(* IEC 61131-3 sources: Summary-ETFA22/ahorn/benchmark/PPU/Scenario3v1_Final, 6 files *)

(* ---- Scenario3v1_Final_Type.st ---- *)
TYPE
    Stamp_states_t : (Green_Lamp , Init , Interstep , Interstep_2 , StampProcess , StampSliderBack , StampSliderForward , Stamp_Init_1 , Stamp_Init_2 , Stamp_Init_3 , Stamp_Init_4 , Start_Stamp , Step0 , Step1 , Step2);
    Magazin_states_t : (Green_Lamp , Init , Interstep , Magazin_Init , Magazin_Init_2 , Slider_Move_Back , Start_Magazin , Step0 , Step1 , convey);
    Crane_states_t : (Crane_Go_Up , Crane_Init , Crane_Init_2 , Crane_Lift_At_Stamp , Crane_Lift_Conveyor , Crane_Lift_Magazin , Crane_Lift_Magazin_Metallic , Crane_Lower , Crane_On_Conveyor , Crane_On_Conveyor_Metallic , Crane_On_Stamp_Metallic , Crane_Turn_Left_From_Stamp , Crane_Turn_Left_Metallic , Crane_Turn_Left_NOT_Metallic , Init , Interstep , Interstep_2 , Interstep_Check_Workpiece , Lower_Crane , Reset_interconnect , Start_Crane , Step0 , Step2 , Suck_At_Stamp , TimeDelay , Turn_Right , Wait_At_Stamp , pause , release , release_Workpiece);
END_TYPE

(* ---- Scenario3v1_Final_Crane.st ---- *)
FUNCTION_BLOCK Crane
    VAR_INPUT  CraneDown : BOOL; END_VAR
    VAR_OUTPUT  CraneLower : BOOL; END_VAR
    VAR_INPUT  CraneOnConveyor : BOOL; END_VAR
    VAR_INPUT  CraneOnMagazin : BOOL; END_VAR
    VAR_INPUT  CranePositionStamp : BOOL; END_VAR
    VAR_INPUT  CraneSucked : BOOL; END_VAR
    VAR_OUTPUT  CraneTurnClockwise : BOOL; END_VAR
    VAR_OUTPUT  CraneTurnCounterclockwise : BOOL; END_VAR
    VAR_INPUT  CraneUp : BOOL; END_VAR
    VAR  Duration1 : TIME := TIME#1s500.0ms; END_VAR
    VAR_INPUT  MagazinCapacitiveSensor : BOOL; END_VAR
    VAR_OUTPUT  MagazinVacuumOff : BOOL; END_VAR
    VAR_OUTPUT  MagazinVacuumOn : BOOL; END_VAR
    VAR  SFCInit : BOOL; END_VAR
    VAR_INPUT  SFCReset : BOOL; END_VAR
    VAR_INPUT  SliderMovedOut : BOOL; END_VAR
    VAR_INPUT  SliderNotMovedOut : BOOL; END_VAR
    VAR_INPUT  StampLowered : BOOL; END_VAR
    VAR_INPUT  StampSliderFilled : BOOL; END_VAR
    VAR_INPUT  StartButtonMagazin : BOOL; END_VAR
    VAR_OUTPUT  StartCommandCrane : BOOL; END_VAR
    VAR_INPUT  StartVar : BOOL; END_VAR
    VAR  TimeDelay_Timer : TON; END_VAR
    VAR  TimeDelay_Timer_Duration : TIME := TIME#50.0ms; END_VAR
    VAR  TimeDelay_Timer_interconnect : BOOL; END_VAR
    VAR  Timer1 : TON; END_VAR
    VAR_INPUT  WorkpieceReady : BOOL; END_VAR
    VAR  State : Crane_states_t; END_VAR
    VAR  Transit : BOOL; END_VAR
    VAR  actualtime1 : TIME; END_VAR
    VAR  interconnect : BOOL; END_VAR
    VAR  interconnectCraneStartCommand : BOOL; END_VAR

    CASE State OF
        Crane_states_t#Crane_Go_Up:
            Transit := FALSE;
            CraneLower := FALSE;
            IF CraneUp THEN
                Transit := TRUE;
                State := Crane_states_t#pause;
            END_IF;

        Crane_states_t#Crane_Init:
            Transit := FALSE;
            CraneLower := TRUE;
            interconnectCraneStartCommand := FALSE;
            IF CraneDown THEN
                Transit := TRUE;
                State := Crane_states_t#Crane_Init_2;
            END_IF;

        Crane_states_t#Crane_Init_2:
            Transit := FALSE;
            CraneLower := FALSE;
            IF CraneUp THEN
                Transit := TRUE;
                State := Crane_states_t#Interstep;
            END_IF;

        Crane_states_t#Crane_Lift_At_Stamp:
            Transit := FALSE;
            CraneLower := FALSE;
            IF CraneUp THEN
                Transit := TRUE;
                State := Crane_states_t#Crane_Turn_Left_From_Stamp;
            END_IF;

        Crane_states_t#Crane_Lift_Conveyor:
            Transit := FALSE;
            CraneLower := FALSE;
            IF TRUE THEN
                Transit := TRUE;
                State := Crane_states_t#Interstep;
            END_IF;

        Crane_states_t#Crane_Lift_Magazin:
            Transit := FALSE;
            CraneLower := FALSE;
            IF CraneUp THEN
                Transit := TRUE;
                State := Crane_states_t#Crane_Turn_Left_NOT_Metallic;
            END_IF;

        Crane_states_t#Crane_Lift_Magazin_Metallic:
            Transit := FALSE;
            CraneLower := FALSE;
            IF CraneUp THEN
                Transit := TRUE;
                State := Crane_states_t#Crane_Turn_Left_Metallic;
            END_IF;

        Crane_states_t#Crane_Lower:
            Transit := FALSE;
            MagazinVacuumOn := TRUE;
            MagazinVacuumOff := FALSE;
            CraneLower := TRUE;
            IF CraneSucked THEN
                Transit := TRUE;
                State := Crane_states_t#Step0;
            END_IF;

        Crane_states_t#Crane_On_Conveyor:
            Transit := FALSE;
            CraneTurnCounterclockwise := FALSE;
            CraneTurnClockwise := FALSE;
            CraneLower := TRUE;
            IF CraneDown THEN
                Transit := TRUE;
                State := Crane_states_t#release;
            END_IF;

        Crane_states_t#Crane_On_Conveyor_Metallic:
            Transit := FALSE;
            CraneTurnCounterclockwise := FALSE;
            CraneTurnClockwise := FALSE;
            CraneLower := TRUE;
            IF CraneDown THEN
                Transit := TRUE;
                State := Crane_states_t#release;
            END_IF;

        Crane_states_t#Crane_On_Stamp_Metallic:
            Transit := FALSE;
            CraneTurnCounterclockwise := FALSE;
            CraneTurnClockwise := FALSE;
            CraneLower := TRUE;
            IF CraneDown THEN
                Transit := TRUE;
                State := Crane_states_t#release_Workpiece;
            END_IF;

        Crane_states_t#Crane_Turn_Left_From_Stamp:
            Transit := FALSE;
            CraneTurnClockwise := TRUE;
            CraneTurnCounterclockwise := FALSE;
            IF CraneOnConveyor THEN
                Transit := TRUE;
                State := Crane_states_t#Crane_On_Conveyor_Metallic;
            END_IF;

        Crane_states_t#Crane_Turn_Left_Metallic:
            Transit := FALSE;
            CraneTurnCounterclockwise := TRUE;
            CraneTurnClockwise := FALSE;
            IF CranePositionStamp THEN
                Transit := TRUE;
                State := Crane_states_t#Crane_On_Stamp_Metallic;
            END_IF;

        Crane_states_t#Crane_Turn_Left_NOT_Metallic:
            Transit := FALSE;
            CraneTurnCounterclockwise := TRUE;
            CraneTurnClockwise := FALSE;
            IF CraneOnConveyor THEN
                Transit := TRUE;
                State := Crane_states_t#Crane_On_Conveyor;
            END_IF;

        Crane_states_t#Init:
            Transit := FALSE;
            IF TRUE THEN
                Transit := TRUE;
                State := Crane_states_t#Start_Crane;
            END_IF;

        Crane_states_t#Interstep:
            Transit := FALSE;
            StartCommandCrane := TRUE;
            IF StartVar THEN
                Transit := TRUE;
                State := Crane_states_t#Interstep_2;
            END_IF;

        Crane_states_t#Interstep_2:
            Transit := FALSE;
            IF SliderMovedOut THEN
                Transit := TRUE;
                State := Crane_states_t#TimeDelay;
            END_IF;

        Crane_states_t#Interstep_Check_Workpiece:
            Transit := FALSE;
            CraneTurnClockwise := FALSE;
            CraneTurnCounterClockwise := FALSE;
            IF WorkpieceReady THEN
                Transit := TRUE;
                State := Crane_states_t#Crane_Lower;
            ELSIF (NOT WorkpieceReady AND NOT StampSliderFilled) THEN
                Transit := TRUE;
                State := Crane_states_t#Step2;
            ELSIF (NOT WorkpieceReady AND StampSliderFilled) THEN
                Transit := TRUE;
                State := Crane_states_t#Wait_At_Stamp;
            END_IF;

        Crane_states_t#Lower_Crane:
            Transit := FALSE;
            CraneLower := TRUE;
            IF CraneDown THEN
                Transit := TRUE;
                State := Crane_states_t#Suck_At_Stamp;
            END_IF;

        Crane_states_t#Reset_interconnect:
            Transit := FALSE;
            interconnect := FALSE;
            Timer1(IN := FALSE, PT := TIME#1.0ms);
            IF SliderMovedOut THEN
                Transit := TRUE;
                State := Crane_states_t#Lower_Crane;
            END_IF;

        Crane_states_t#Start_Crane:
            Transit := FALSE;
            CraneLower := FALSE;
            MagazinVacuumOff := TRUE;
            MagazinVacuumOn := FALSE;
            CraneTurnCounterclockwise := FALSE;
            CraneTurnClockwise := FALSE;
            StartVar := FALSE;
            StartCommandCrane := FALSE;
            IF (StartButtonMagazin = TRUE) THEN
                interconnectCraneStartCommand := TRUE;
            END_IF;
            IF interconnectCraneStartCommand THEN
                Transit := TRUE;
                State := Crane_states_t#Crane_Init;
            END_IF;

        Crane_states_t#Step0:
            Transit := FALSE;
            IF NOT MagazinCapacitiveSensor THEN
                Transit := TRUE;
                State := Crane_states_t#Crane_Lift_Magazin;
            ELSIF MagazinCapacitiveSensor THEN
                Transit := TRUE;
                State := Crane_states_t#Crane_Lift_Magazin_Metallic;
            END_IF;

        Crane_states_t#Step2:
            Transit := FALSE;
            IF TRUE THEN
                Transit := TRUE;
                State := Crane_states_t#Start_Crane;
            END_IF;

        Crane_states_t#Suck_At_Stamp:
            Transit := FALSE;
            MagazinVacuumOn := TRUE;
            MagazinVacuumOff := FALSE;
            IF CraneSucked THEN
                Transit := TRUE;
                State := Crane_states_t#Crane_Lift_At_Stamp;
            END_IF;

        Crane_states_t#TimeDelay:
            Transit := FALSE;
            TimeDelay_Timer(IN := TRUE, PT := TimeDelay_Timer_Duration);
            TimeDelay_Timer_interconnect := TimeDelay_Timer.Q;
            IF TimeDelay_Timer_interconnect THEN
                Transit := TRUE;
                State := Crane_states_t#Turn_Right;
            END_IF;

        Crane_states_t#Turn_Right:
            Transit := FALSE;
            CraneTurnClockwise := TRUE;
            CraneTurnCounterclockwise := FALSE;
            IF CraneOnMagazin THEN
                Transit := TRUE;
                State := Crane_states_t#Interstep_Check_Workpiece;
            END_IF;

        Crane_states_t#Wait_At_Stamp:
            Transit := FALSE;
            IF TRUE THEN
                Transit := TRUE;
                State := Crane_states_t#pause;
            END_IF;

        Crane_states_t#pause:
            Transit := FALSE;
            Timer1(IN := CraneUp, PT := Duration1);
            interconnect := Timer1.Q;
            IF interconnect THEN
                Transit := TRUE;
                State := Crane_states_t#Reset_interconnect;
            END_IF;

        Crane_states_t#release:
            Transit := FALSE;
            MagazinVacuumOff := TRUE;
            MagazinVacuumOn := FALSE;
            IF TRUE THEN
                Transit := TRUE;
                State := Crane_states_t#Crane_Lift_Conveyor;
            END_IF;

        Crane_states_t#release_Workpiece:
            Transit := FALSE;
            MagazinVacuumOff := TRUE;
            MagazinVacuumOn := FALSE;
            IF TRUE THEN
                Transit := TRUE;
                State := Crane_states_t#Crane_Go_Up;
            END_IF;
    END_CASE;
END_FUNCTION_BLOCK

(* ---- Scenario3v1_Final_Magazin.st ---- *)
FUNCTION_BLOCK Magazin
    VAR_INPUT  CraneDown : BOOL; END_VAR
    VAR_OUTPUT  CraneLower : BOOL; END_VAR
    VAR_INPUT  CraneOnConveyor : BOOL; END_VAR
    VAR_INPUT  CraneOnMagazin : BOOL; END_VAR
    VAR_INPUT  CraneSucked : BOOL; END_VAR
    VAR_OUTPUT  CraneTurnClockwise : BOOL; END_VAR
    VAR_OUTPUT  CraneTurnCounterclockwise : BOOL; END_VAR
    VAR_INPUT  CraneUp : BOOL; END_VAR
    VAR_OUTPUT  MagazinGreenLamp : BOOL; END_VAR
    VAR_OUTPUT  MagazinSlider : BOOL; END_VAR
    VAR_OUTPUT  MagazinVacuumOff : BOOL; END_VAR
    VAR_OUTPUT  MagazinVacuumOn : BOOL; END_VAR
    VAR_OUTPUT  MagazinWhiteLamp : BOOL; END_VAR
    VAR  SFCInit : BOOL; END_VAR
    VAR_INPUT  SFCReset : BOOL; END_VAR
    VAR_INPUT  SliderMovedOut : BOOL; END_VAR
    VAR_INPUT  SliderNotMovedOut : BOOL; END_VAR
    VAR_INPUT  StartButtonMagazin : BOOL; END_VAR
    VAR_OUTPUT  StartCommandMagazin : BOOL; END_VAR
    VAR_INPUT  StartVar : BOOL; END_VAR
    VAR_INPUT  WorkpieceReady : BOOL; END_VAR
    VAR  State : Magazin_states_t; END_VAR
    VAR Transit : BOOL; END_VAR
    VAR  interconnectMagazinStartCommand : BOOL; END_VAR

    CASE State OF
        Magazin_states_t#Green_Lamp:

            (* begin(onEntry) *)
           Transit := FALSE;
            (* end(onEntry) *)
            (* begin(onActive) *)
            MagazinGreenLamp := TRUE;
            interconnectMagazinStartCommand := FALSE;
            (* end(onActive) *)
            (* begin(transition) *)
            IF TRUE THEN
               Transit := TRUE;
                State := Magazin_states_t#Magazin_Init;
            END_IF;
            (* end(transition) *)
            (* begin(onExit) *)
            (* end(onExit) *)
            (* end(State) *)

        Magazin_states_t#Init:

            (* begin(onEntry) *)
           Transit := FALSE;
            (* end(onEntry) *)
            (* begin(onActive) *)
            (* end(onActive) *)
            (* begin(transition) *)
            IF TRUE THEN
               Transit := TRUE;
                State := Magazin_states_t#Start_Magazin;
            END_IF;
            (* end(transition) *)
            (* begin(onExit) *)
            (* end(onExit) *)
            (* end(State) *)

        Magazin_states_t#Interstep:

            (* begin(onEntry) *)
           Transit := FALSE;
            (* end(onEntry) *)
            (* begin(onActive) *)
            StartCommandMagazin := TRUE;
            (* end(onActive) *)
            (* begin(transition) *)
            IF StartVar THEN
               Transit := TRUE;
                State := Magazin_states_t#convey;
            END_IF;
            (* end(transition) *)
            (* begin(onExit) *)
            (* end(onExit) *)
            (* end(State) *)

        Magazin_states_t#Magazin_Init:

            (* begin(onEntry) *)
           Transit := FALSE;
            (* end(onEntry) *)
            (* begin(onActive) *)
            MagazinSlider := TRUE;
            (* end(onActive) *)
            (* begin(transition) *)
            IF TRUE THEN
               Transit := TRUE;
                State := Magazin_states_t#Magazin_Init_2;
            END_IF;
            (* end(transition) *)
            (* begin(onExit) *)
            (* end(onExit) *)
            (* end(State) *)

        Magazin_states_t#Magazin_Init_2:

            (* begin(onEntry) *)
           Transit := FALSE;
            (* end(onEntry) *)
            (* begin(onActive) *)
            MagazinSlider := FALSE;
            (* end(onActive) *)
            (* begin(transition) *)
            IF TRUE THEN
               Transit := TRUE;
                State := Magazin_states_t#Interstep;
            END_IF;
            (* end(transition) *)
            (* begin(onExit) *)
            (* end(onExit) *)
            (* end(State) *)

        Magazin_states_t#Slider_Move_Back:

            (* begin(onEntry) *)
           Transit := FALSE;
            (* end(onEntry) *)
            (* begin(onActive) *)
            IF ((SliderMovedOut = TRUE) AND (SliderNotMovedOut = FALSE)) THEN
                MagazinSlider := FALSE;
            END_IF;
            (* end(onActive) *)
            (* begin(transition) *)
            IF CraneUp THEN
               Transit := TRUE;
                State := Magazin_states_t#Step1;
            END_IF;
            (* end(transition) *)
            (* begin(onExit) *)
            (* end(onExit) *)
            (* end(State) *)

        Magazin_states_t#Start_Magazin:

            (* begin(onEntry) *)
           Transit := FALSE;
            (* end(onEntry) *)
            (* begin(onActive) *)
            MagazinSlider := FALSE;
            MagazinGreenLamp := FALSE;
            StartVar := FALSE;
            StartCommandMagazin := FALSE;
            IF (StartButtonMagazin = TRUE) THEN
                interconnectMagazinStartCommand := TRUE;
            END_IF;
            (* end(onActive) *)
            (* begin(transition) *)
            IF interconnectMagazinStartCommand THEN
               Transit := TRUE;
                State := Magazin_states_t#Green_Lamp;
            END_IF;
            (* end(transition) *)
            (* begin(onExit) *)
            (* end(onExit) *)
            (* end(State) *)

        Magazin_states_t#Step0:

            (* begin(onEntry) *)
           Transit := FALSE;
            (* end(onEntry) *)
            (* begin(onActive) *)
            (* end(onActive) *)
            (* begin(transition) *)
            IF CraneDown THEN
               Transit := TRUE;
                State := Magazin_states_t#Slider_Move_Back;
            END_IF;
            (* end(transition) *)
            (* begin(onExit) *)
            (* end(onExit) *)
            (* end(State) *)

        Magazin_states_t#Step1:

            (* begin(onEntry) *)
           Transit := FALSE;
            (* end(onEntry) *)
            (* begin(onActive) *)
            (* end(onActive) *)
            (* begin(transition) *)
            IF CraneOnConveyor THEN
               Transit := TRUE;
                State := Magazin_states_t#Interstep;
            END_IF;
            (* end(transition) *)
            (* begin(onExit) *)
            (* end(onExit) *)
            (* end(State) *)

        Magazin_states_t#convey:

            (* begin(onEntry) *)
           Transit := FALSE;
            (* end(onEntry) *)
            (* begin(onActive) *)
            IF SliderNotMovedOut THEN
                MagazinSlider := TRUE;
            END_IF;
            (* end(onActive) *)
            (* begin(transition) *)
            IF CraneOnMagazin THEN
               Transit := TRUE;
                State := Magazin_states_t#Step0;
            END_IF;
            (* end(transition) *)
            (* begin(onExit) *)
            (* end(onExit) *)
            (* end(State) *)

            END_CASE;
END_FUNCTION_BLOCK

(* ---- Scenario3v1_Final_Stamp.st ---- *)
FUNCTION_BLOCK Stamp
    VAR_INPUT  CraneDown : BOOL; END_VAR (*Irwxp*)
    VAR_INPUT  CraneOnConveyor : BOOL; END_VAR (*Irwxp*)
    VAR_INPUT  CranePositionStamp : BOOL; END_VAR (*Irwxp*)
    VAR_INPUT  CraneSucked : BOOL; END_VAR (*Irwxp*)
    VAR_INPUT  CraneUp : BOOL; END_VAR (*Irwxp*)
    VAR  Duration : TIME := TIME#500.0ms; END_VAR (*Lrwxp*)
    VAR  SFCInit : BOOL; END_VAR (*Lrwxp*)
    VAR_INPUT  SFCReset : BOOL; END_VAR (*Irwxp*)
    VAR_OUTPUT  StampGreenLamp : BOOL; END_VAR (*Orwxp*)
    VAR_INPUT  StampLowered : BOOL; END_VAR (*Irwxp*)
    VAR_OUTPUT  StampPressure : BOOL; END_VAR (*Orwxp*)
    VAR_OUTPUT  StampPusher : BOOL; END_VAR (*Orwxp*)
    VAR_INPUT  StampSliderFilled : BOOL; END_VAR (*Irwxp*)
    VAR_OUTPUT  StampSliderMovedIn : BOOL; END_VAR (*Orwxp*)
    VAR_OUTPUT  StampSliderMovedOut : BOOL; END_VAR (*Orwxp*)
    VAR_INPUT  StampSliderSensorMovedIn : BOOL; END_VAR (*Irwxp*)
    VAR_INPUT  StampSliderSensorMovedOut : BOOL; END_VAR (*Irwxp*)
    VAR_INPUT  StampStartButton : BOOL; END_VAR (*Irwxp*)
    VAR_INPUT  StampUp : BOOL; END_VAR (*Irwxp*)
    VAR_OUTPUT  StampWhiteLamp : BOOL; END_VAR (*Orwxp*)
    VAR_OUTPUT  StartCommandStamp : BOOL; END_VAR (*Orwxp*)
    VAR_INPUT  StartVar : BOOL; END_VAR (*Irwxp*)
    VAR  Timer : TON; END_VAR (*Lrwxp*)
    VAR  State : Stamp_states_t; END_VAR (*Lrwxp*)
    VAR  Transit : BOOL; END_VAR (*Lrwxp*)
    VAR  interconnect : BOOL; END_VAR (*Lrwxp*)
    VAR  interconnectStampStartCommand : BOOL; END_VAR (*Lrwxp*)

    CASE State OF
        Stamp_states_t#Green_Lamp:

            (* begin(onEntry) *)
            Transit := FALSE;
            (* end(onEntry) *)
            (* begin(onActive) *)
            StampGreenLamp := TRUE;
            interconnectStampStartCommand := FALSE;
            (* end(onActive) *)
            (* begin(transition) *)
            IF TRUE THEN
                Transit := TRUE;
                State := Stamp_states_t#Stamp_Init_1;
            END_IF;
            (* end(transition) *)
            (* begin(onExit) *)
            (* end(onExit) *)
            (* end(State) *)

        Stamp_states_t#Init:

            (* begin(onEntry) *)
            Transit := FALSE;
            (* end(onEntry) *)
            (* begin(onActive) *)
            (* end(onActive) *)
            (* begin(transition) *)
            IF TRUE THEN
                Transit := TRUE;
                State := Stamp_states_t#Start_Stamp;
            END_IF;
            (* end(transition) *)
            (* begin(onExit) *)
            (* end(onExit) *)
            (* end(State) *)

        Stamp_states_t#Interstep:

            (* begin(onEntry) *)
            Transit := FALSE;
            (* end(onEntry) *)
            (* begin(onActive) *)
            StartCommandStamp := TRUE;
            (* end(onActive) *)
            (* begin(transition) *)
            IF StartVar THEN
                Transit := TRUE;
                State := Stamp_states_t#Interstep_2;
            END_IF;
            (* end(transition) *)
            (* begin(onExit) *)
            (* end(onExit) *)
            (* end(State) *)

        Stamp_states_t#Interstep_2:

            (* begin(onEntry) *)
            Transit := FALSE;
            (* end(onEntry) *)
            (* begin(onActive) *)
            (* end(onActive) *)
            (* begin(transition) *)
            IF StampSliderFilled THEN
                Transit := TRUE;
                State := Stamp_states_t#Step0;
            END_IF;
            (* end(transition) *)
            (* begin(onExit) *)
            (* end(onExit) *)
            (* end(State) *)

        Stamp_states_t#StampProcess:

            (* begin(onEntry) *)
            Transit := FALSE;
            (* end(onEntry) *)
            (* begin(onActive) *)
            StampSliderMovedIn := FALSE;
            StampPusher := TRUE;
            (* end(onActive) *)
            (* begin(transition) *)
            IF StampLowered THEN
                Transit := TRUE;
                State := Stamp_states_t#Step1;
            END_IF;
            (* end(transition) *)
            (* begin(onExit) *)
            (* end(onExit) *)
            (* end(State) *)

        Stamp_states_t#StampSliderBack:

            (* begin(onEntry) *)
            Transit := FALSE;
            (* end(onEntry) *)
            (* begin(onActive) *)
            StampSliderMovedIn := TRUE;
            StampSliderMovedOut := FALSE;
            (* end(onActive) *)
            (* begin(transition) *)
            IF StampSliderSensorMovedIn THEN
                Transit := TRUE;
                State := Stamp_states_t#StampProcess;
            END_IF;
            (* end(transition) *)
            (* begin(onExit) *)
            (* end(onExit) *)
            (* end(State) *)

        Stamp_states_t#StampSliderForward:

            (* begin(onEntry) *)
            Transit := FALSE;
            (* end(onEntry) *)
            (* begin(onActive) *)
            StampPusher := FALSE;
            StampSliderMovedOut := TRUE;
            IF ((StampLowered = FALSE) AND (StampUp = TRUE)) THEN
                interconnect := FALSE;
            END_IF;
            Timer(IN := FALSE, PT := TIME#1.0ms);
            (* end(onActive) *)
            (* begin(transition) *)
            IF StampSliderMovedOut THEN
                Transit := TRUE;
                State := Stamp_states_t#Step2;
            END_IF;
            (* end(transition) *)
            (* begin(onExit) *)
            (* end(onExit) *)
            (* end(State) *)

        Stamp_states_t#Stamp_Init_1:

            (* begin(onEntry) *)
            Transit := FALSE;
            (* end(onEntry) *)
            (* begin(onActive) *)
            StampSliderMovedIn := TRUE;
            StampSliderMovedOut := FALSE;
            (* end(onActive) *)
            (* begin(transition) *)
            IF StampSliderSensorMovedIn THEN
                Transit := TRUE;
                State := Stamp_states_t#Stamp_Init_2;
            END_IF;
            (* end(transition) *)
            (* begin(onExit) *)
            (* end(onExit) *)
            (* end(State) *)

        Stamp_states_t#Stamp_Init_2:

            (* begin(onEntry) *)
            Transit := FALSE;
            (* end(onEntry) *)
            (* begin(onActive) *)
            StampSliderMovedIn := FALSE;
            StampSliderMovedOut := TRUE;
            (* end(onActive) *)
            (* begin(transition) *)
            IF StampSliderSensorMovedOut THEN
                Transit := TRUE;
                State := Stamp_states_t#Stamp_Init_3;
            END_IF;
            (* end(transition) *)
            (* begin(onExit) *)
            (* end(onExit) *)
            (* end(State) *)

        Stamp_states_t#Stamp_Init_3:

            (* begin(onEntry) *)
            Transit := FALSE;
            (* end(onEntry) *)
            (* begin(onActive) *)
            StampPusher := TRUE;
            (* end(onActive) *)
            (* begin(transition) *)
            IF StampLowered THEN
                Transit := TRUE;
                State := Stamp_states_t#Stamp_Init_4;
            END_IF;
            (* end(transition) *)
            (* begin(onExit) *)
            (* end(onExit) *)
            (* end(State) *)

        Stamp_states_t#Stamp_Init_4:

            (* begin(onEntry) *)
            Transit := FALSE;
            (* end(onEntry) *)
            (* begin(onActive) *)
            StampPusher := FALSE;
            (* end(onActive) *)
            (* begin(transition) *)
            IF StampUp THEN
                Transit := TRUE;
                State := Stamp_states_t#Interstep;
            END_IF;
            (* end(transition) *)
            (* begin(onExit) *)
            (* end(onExit) *)
            (* end(State) *)

        Stamp_states_t#Start_Stamp:

            (* begin(onEntry) *)
            Transit := FALSE;
            (* end(onEntry) *)
            (* begin(onActive) *)
            StampSliderMovedOut := FALSE;
            StampSliderMovedIn := FALSE;
            StampPusher := FALSE;
            StampGreenLamp := FALSE;
            StampPressure := FALSE;
            StartCommandStamp := FALSE;
            IF (StampStartButton = TRUE) THEN
                interconnectStampStartCommand := TRUE;
            END_IF;
            (* end(onActive) *)
            (* begin(transition) *)
            IF interconnectStampStartCommand THEN
                Transit := TRUE;
                State := Stamp_states_t#Green_Lamp;
            END_IF;
            (* end(transition) *)
            (* begin(onExit) *)
            (* end(onExit) *)
            (* end(State) *)

        Stamp_states_t#Step0:

            (* begin(onEntry) *)
            Transit := FALSE;
            (* end(onEntry) *)
            (* begin(onActive) *)
            (* end(onActive) *)
            (* begin(transition) *)
            IF CraneUp THEN
                Transit := TRUE;
                State := Stamp_states_t#StampSliderBack;
            END_IF;
            (* end(transition) *)
            (* begin(onExit) *)
            (* end(onExit) *)
            (* end(State) *)

        Stamp_states_t#Step1:

            (* begin(onEntry) *)
            Transit := FALSE;
            (* end(onEntry) *)
            (* begin(onActive) *)
            Timer(IN := StampLowered, PT := T#500ms);
            interconnect := Timer.Q;
            (* end(onActive) *)
            (* begin(transition) *)
            IF interconnect THEN
                Transit := TRUE;
                State := Stamp_states_t#StampSliderForward;
            END_IF;
            (* end(transition) *)
            (* begin(onExit) *)
            (* end(onExit) *)
            (* end(State) *)

        Stamp_states_t#Step2:

            (* begin(onEntry) *)
            Transit := FALSE;
            (* end(onEntry) *)
            (* begin(onActive) *)
            (* end(onActive) *)
            (* begin(transition) *)
            IF CraneOnConveyor THEN
                Transit := TRUE;
                State := Stamp_states_t#Interstep;
            END_IF;
            (* end(transition) *)
            (* begin(onExit) *)
            (* end(onExit) *)
            (* end(State) *)

            END_CASE;
END_FUNCTION_BLOCK

(* ---- Scenario3v1_Final.st ---- *)
PROGRAM Main

VAR  Actuator_AnalogCranePressure : INT; END_VAR (*Lrwxp*)
VAR  Actuator_CraneLower : BOOL; END_VAR (*Lrwxp*)
VAR  Actuator_CraneTurnClockwise : BOOL; END_VAR (*Lrwxp*)
VAR  Actuator_CraneTurnCounterclockwise : BOOL; END_VAR (*Lrwxp*)
VAR  Actuator_MagazinGreenLamp : BOOL; END_VAR (*Lrwxp*)
VAR  Actuator_MagazinSlider : BOOL; END_VAR (*Lrwxp*)
VAR  Actuator_MagazinVacuumOff : BOOL; END_VAR (*Lrwxp*)
VAR  Actuator_MagazinVacuumOn : BOOL; END_VAR (*Lrwxp*)
VAR  Actuator_MagazinWhiteLamp : BOOL; END_VAR (*Lrwxp*)
VAR  Actuator_SomeActuator : BOOL; END_VAR (*Lrwxp*)
VAR  Actuator_StampGreenLamp : BOOL; END_VAR (*Lrwxp*)
VAR  Actuator_StampPusher : BOOL; END_VAR (*Lrwxp*)
VAR  Actuator_StampSliderMovedIn : BOOL; END_VAR (*Lrwxp*)
VAR  Actuator_StampSliderMovedOut : BOOL; END_VAR (*Lrwxp*)
VAR  Actuator_StampWhiteLamp : BOOL; END_VAR (*Lrwxp*)
VAR  Crane : Crane; END_VAR (*Lrwxp*)
VAR  Mag : Magazin; END_VAR (*Lrwxp*)
VAR  Sensor_CraneDown : BOOL; END_VAR (*Lrwxp*)
VAR  Sensor_CraneOnConveyor : BOOL; END_VAR (*Lrwxp*)
VAR  Sensor_CraneOnMagazin : BOOL; END_VAR (*Lrwxp*)
VAR  Sensor_CranePosition : BOOL; END_VAR (*Lrwxp*)
VAR  Sensor_CranePositionStamp : BOOL; END_VAR (*Lrwxp*)
VAR  Sensor_CraneSucked : BOOL; END_VAR (*Lrwxp*)
VAR  Sensor_CraneUp : BOOL; END_VAR (*Lrwxp*)
VAR  Sensor_MagazinCapacitiveSensor : BOOL; END_VAR (*Lrwxp*)
VAR  Sensor_MagazinEmergencyStop : BOOL; END_VAR (*Lrwxp*)
VAR  Sensor_MagazinOpticalSensor : BOOL; END_VAR (*Lrwxp*)
VAR  Sensor_MagazinSwitchManuellAutomatic : BOOL; END_VAR (*Lrwxp*)
VAR  Sensor_SliderMovedOut : BOOL; END_VAR (*Lrwxp*)
VAR  Sensor_SliderNotMovedOut : BOOL; END_VAR (*Lrwxp*)
VAR  Sensor_StampEmergencyStop : BOOL; END_VAR (*Lrwxp*)
VAR  Sensor_StampLowered : BOOL; END_VAR (*Lrwxp*)
VAR  Sensor_StampSliderFilled : BOOL; END_VAR (*Lrwxp*)
VAR  Sensor_StampSliderSensorMovedIn : BOOL; END_VAR (*Lrwxp*)
VAR  Sensor_StampSliderSensorMovedOut : BOOL; END_VAR (*Lrwxp*)
VAR  Sensor_StampStartButton : BOOL; END_VAR (*Lrwxp*)
VAR  Sensor_StampSwitchManuellAutomatic : BOOL; END_VAR (*Lrwxp*)
VAR  Sensor_StampUp : BOOL; END_VAR (*Lrwxp*)
VAR  Sensor_StartButtonMagazin : BOOL; END_VAR (*Lrwxp*)
VAR  Sensor_WorkpieceReady : BOOL; END_VAR (*Lrwxp*)
VAR  Stamp : Stamp; END_VAR (*Lrwxp*)
Mag.SliderNotMovedOut := Sensor_SliderNotMovedOut;
Mag.SliderMovedOut := Sensor_SliderMovedOut;
Mag.CraneOnMagazin := Sensor_CraneOnMagazin;
Mag.CraneDown := Sensor_CraneDown;
Mag.CraneUp := Sensor_CraneUp;
Mag.CraneOnConveyor := Sensor_CraneOnConveyor;
Mag.WorkpieceReady := Sensor_WorkpieceReady;
Mag.StartButtonMagazin := Sensor_StartButtonMagazin;
Actuator_MagazinSlider := Mag.MagazinSlider;
Actuator_MagazinGreenLamp := Mag.MagazinGreenLamp;
Crane.CraneUp := Sensor_CraneUp;
Crane.CraneOnConveyor := Sensor_CraneOnConveyor;
Crane.CraneDown := Sensor_CraneDown;
Crane.CraneSucked := Sensor_CraneSucked;
Crane.CraneOnMagazin := Sensor_CraneOnMagazin;
Crane.MagazinCapacitiveSensor := Sensor_MagazinCapacitiveSensor;
Crane.CranePositionStamp := Sensor_CranePositionStamp;
Crane.SliderMovedOut := Sensor_SliderMovedOut;
Crane.WorkpieceReady := Sensor_WorkpieceReady;
Crane.StampSliderFilled := Sensor_StampSliderFilled;
Crane.SliderMovedOut := Sensor_SliderMovedOut;
Crane.StartButtonMagazin := Sensor_StartButtonMagazin;
Actuator_CraneTurnCounterclockwise := Crane.CraneTurnCounterclockwise;
Actuator_CraneTurnClockwise := Crane.CraneTurnClockwise;
Actuator_CraneLower := Crane.CraneLower;
Actuator_MagazinVacuumOff := Crane.MagazinVacuumOff;
Actuator_MagazinVacuumOn := Crane.MagazinVacuumOn;
Stamp.StampSliderSensorMovedOut := Sensor_StampSliderSensorMovedOut;
Stamp.StampSliderSensorMovedIn := Sensor_StampSliderSensorMovedIn;
Stamp.StampSliderFilled := Sensor_StampSliderFilled;
Stamp.StampUp := Sensor_StampUp;
Stamp.StampLowered := Sensor_StampLowered;
Stamp.CraneDown := Sensor_CraneDown;
Stamp.CraneUp := Sensor_CraneUp;
Stamp.CraneSucked := Sensor_CraneSucked;
Stamp.CranePositionStamp := Sensor_CranePositionStamp;
Stamp.CraneOnConveyor := Sensor_CraneOnConveyor;
Stamp.StampStartButton := Sensor_StampStartButton;
Actuator_StampSliderMovedOut := Stamp.StampSliderMovedOut;
Actuator_StampSliderMovedIn := Stamp.StampSliderMovedIn;
Actuator_StampWhiteLamp := Stamp.StampWhiteLamp;
Actuator_StampPusher := Stamp.StampPusher;
Actuator_StampGreenLamp := Stamp.StampGreenLamp;
Actuator_AnalogCranePressure := INT#6000;
IF (Sensor_StampEmergencyStop AND Sensor_MagazinEmergencyStop) THEN
    Mag();
    Crane();
    Stamp();
    IF (Actuator_MagazinGreenLamp AND Actuator_StampGreenLamp) THEN
        IF ((Stamp.StartCommandStamp AND Crane.StartCommandCrane) AND Mag.StartCommandMagazin) THEN
            Crane.StartVar := TRUE;
            Mag.StartVar := TRUE;
            Stamp.StartVar := TRUE;
        END_IF;
    END_IF;
    Crane.SFCReset := FALSE;
    Mag.SFCReset := FALSE;
    Stamp.SFCReset := FALSE;
ELSIF (NOT Sensor_StampEmergencyStop OR NOT Sensor_MagazinEmergencyStop) THEN
    Actuator_MagazinSlider := FALSE;
    Actuator_CraneLower := FALSE;
    Actuator_MagazinVacuumOn := FALSE;
    Actuator_MagazinVacuumOff := TRUE;
    Actuator_MagazinGreenLamp := FALSE;
    Actuator_CraneTurnCounterclockwise := FALSE;
    Actuator_CraneTurnClockwise := FALSE;
    Actuator_StampSliderMovedOut := TRUE;
    Actuator_StampSliderMovedIn := FALSE;
    Actuator_StampGreenLamp := FALSE;
    Actuator_StampPusher := FALSE;
    Actuator_AnalogCranePressure := INT#0;
    Crane.SFCReset := TRUE;
    Mag.SFCReset := TRUE;
    Stamp.SFCReset := TRUE;
    Crane.StartVar := FALSE;
    Mag.StartVar := FALSE;
    Stamp.StartVar := FALSE;
END_IF;
END_PROGRAM

FUNCTION_BLOCK Crane
    VAR_INPUT  CraneDown : BOOL; END_VAR
    VAR_OUTPUT  CraneLower : BOOL; END_VAR
    VAR_INPUT  CraneOnConveyor : BOOL; END_VAR
    VAR_INPUT  CraneOnMagazin : BOOL; END_VAR
    VAR_INPUT  CranePositionStamp : BOOL; END_VAR
    VAR_INPUT  CraneSucked : BOOL; END_VAR
    VAR_OUTPUT  CraneTurnClockwise : BOOL; END_VAR
    VAR_OUTPUT  CraneTurnCounterclockwise : BOOL; END_VAR
    VAR_INPUT  CraneUp : BOOL; END_VAR
    VAR  Duration1 : TIME := TIME#1s500.0ms; END_VAR
    VAR_INPUT  MagazinCapacitiveSensor : BOOL; END_VAR
    VAR_OUTPUT  MagazinVacuumOff : BOOL; END_VAR
    VAR_OUTPUT  MagazinVacuumOn : BOOL; END_VAR
    VAR  SFCInit : BOOL; END_VAR
    VAR_INPUT  SFCReset : BOOL; END_VAR
    VAR_INPUT  SliderMovedOut : BOOL; END_VAR
    VAR_INPUT  SliderNotMovedOut : BOOL; END_VAR
    VAR_INPUT  StampLowered : BOOL; END_VAR
    VAR_INPUT  StampSliderFilled : BOOL; END_VAR
    VAR_INPUT  StartButtonMagazin : BOOL; END_VAR
    VAR_OUTPUT  StartCommandCrane : BOOL; END_VAR
    VAR_INPUT  StartVar : BOOL; END_VAR
    VAR  TimeDelay_Timer : TON; END_VAR
    VAR  TimeDelay_Timer_Duration : TIME := TIME#50.0ms; END_VAR
    VAR  TimeDelay_Timer_interconnect : BOOL; END_VAR
    VAR  Timer1 : TON; END_VAR
    VAR_INPUT  WorkpieceReady : BOOL; END_VAR
    VAR  State : Crane_states_t; END_VAR
    VAR  Transit : BOOL; END_VAR
    VAR  actualtime1 : TIME; END_VAR
    VAR  interconnect : BOOL; END_VAR
    VAR  interconnectCraneStartCommand : BOOL; END_VAR

    CASE State OF
        Crane_states_t#Crane_Go_Up:
            Transit := FALSE;
            CraneLower := FALSE;
            IF CraneUp THEN
                Transit := TRUE;
                State := Crane_states_t#pause;
            END_IF;

        Crane_states_t#Crane_Init:
            Transit := FALSE;
            CraneLower := TRUE;
            interconnectCraneStartCommand := FALSE;
            IF CraneDown THEN
                Transit := TRUE;
                State := Crane_states_t#Crane_Init_2;
            END_IF;

        Crane_states_t#Crane_Init_2:
            Transit := FALSE;
            CraneLower := FALSE;
            IF CraneUp THEN
                Transit := TRUE;
                State := Crane_states_t#Interstep;
            END_IF;

        Crane_states_t#Crane_Lift_At_Stamp:
            Transit := FALSE;
            CraneLower := FALSE;
            IF CraneUp THEN
                Transit := TRUE;
                State := Crane_states_t#Crane_Turn_Left_From_Stamp;
            END_IF;

        Crane_states_t#Crane_Lift_Conveyor:
            Transit := FALSE;
            CraneLower := FALSE;
            IF TRUE THEN
                Transit := TRUE;
                State := Crane_states_t#Interstep;
            END_IF;

        Crane_states_t#Crane_Lift_Magazin:
            Transit := FALSE;
            CraneLower := FALSE;
            IF CraneUp THEN
                Transit := TRUE;
                State := Crane_states_t#Crane_Turn_Left_NOT_Metallic;
            END_IF;

        Crane_states_t#Crane_Lift_Magazin_Metallic:
            Transit := FALSE;
            CraneLower := FALSE;
            IF CraneUp THEN
                Transit := TRUE;
                State := Crane_states_t#Crane_Turn_Left_Metallic;
            END_IF;

        Crane_states_t#Crane_Lower:
            Transit := FALSE;
            MagazinVacuumOn := TRUE;
            MagazinVacuumOff := FALSE;
            CraneLower := TRUE;
            IF CraneSucked THEN
                Transit := TRUE;
                State := Crane_states_t#Step0;
            END_IF;

        Crane_states_t#Crane_On_Conveyor:
            Transit := FALSE;
            CraneTurnCounterclockwise := FALSE;
            CraneTurnClockwise := FALSE;
            CraneLower := TRUE;
            IF CraneDown THEN
                Transit := TRUE;
                State := Crane_states_t#release;
            END_IF;

        Crane_states_t#Crane_On_Conveyor_Metallic:
            Transit := FALSE;
            CraneTurnCounterclockwise := FALSE;
            CraneTurnClockwise := FALSE;
            CraneLower := TRUE;
            IF CraneDown THEN
                Transit := TRUE;
                State := Crane_states_t#release;
            END_IF;

        Crane_states_t#Crane_On_Stamp_Metallic:
            Transit := FALSE;
            CraneTurnCounterclockwise := FALSE;
            CraneTurnClockwise := FALSE;
            CraneLower := TRUE;
            IF CraneDown THEN
                Transit := TRUE;
                State := Crane_states_t#release_Workpiece;
            END_IF;

        Crane_states_t#Crane_Turn_Left_From_Stamp:
            Transit := FALSE;
            CraneTurnClockwise := TRUE;
            CraneTurnCounterclockwise := FALSE;
            IF CraneOnConveyor THEN
                Transit := TRUE;
                State := Crane_states_t#Crane_On_Conveyor_Metallic;
            END_IF;

        Crane_states_t#Crane_Turn_Left_Metallic:
            Transit := FALSE;
            CraneTurnCounterclockwise := TRUE;
            CraneTurnClockwise := FALSE;
            IF CranePositionStamp THEN
                Transit := TRUE;
                State := Crane_states_t#Crane_On_Stamp_Metallic;
            END_IF;

        Crane_states_t#Crane_Turn_Left_NOT_Metallic:
            Transit := FALSE;
            CraneTurnCounterclockwise := TRUE;
            CraneTurnClockwise := FALSE;
            IF CraneOnConveyor THEN
                Transit := TRUE;
                State := Crane_states_t#Crane_On_Conveyor;
            END_IF;

        Crane_states_t#Init:
            Transit := FALSE;
            IF TRUE THEN
                Transit := TRUE;
                State := Crane_states_t#Start_Crane;
            END_IF;

        Crane_states_t#Interstep:
            Transit := FALSE;
            StartCommandCrane := TRUE;
            IF StartVar THEN
                Transit := TRUE;
                State := Crane_states_t#Interstep_2;
            END_IF;

        Crane_states_t#Interstep_2:
            Transit := FALSE;
            IF SliderMovedOut THEN
                Transit := TRUE;
                State := Crane_states_t#TimeDelay;
            END_IF;

        Crane_states_t#Interstep_Check_Workpiece:
            Transit := FALSE;
            CraneTurnClockwise := FALSE;
            CraneTurnCounterClockwise := FALSE;
            IF WorkpieceReady THEN
                Transit := TRUE;
                State := Crane_states_t#Crane_Lower;
            ELSIF (NOT WorkpieceReady AND NOT StampSliderFilled) THEN
                Transit := TRUE;
                State := Crane_states_t#Step2;
            ELSIF (NOT WorkpieceReady AND StampSliderFilled) THEN
                Transit := TRUE;
                State := Crane_states_t#Wait_At_Stamp;
            END_IF;

        Crane_states_t#Lower_Crane:
            Transit := FALSE;
            CraneLower := TRUE;
            IF CraneDown THEN
                Transit := TRUE;
                State := Crane_states_t#Suck_At_Stamp;
            END_IF;

        Crane_states_t#Reset_interconnect:
            Transit := FALSE;
            interconnect := FALSE;
            Timer1(IN := FALSE, PT := TIME#1.0ms);
            IF SliderMovedOut THEN
                Transit := TRUE;
                State := Crane_states_t#Lower_Crane;
            END_IF;

        Crane_states_t#Start_Crane:
            Transit := FALSE;
            CraneLower := FALSE;
            MagazinVacuumOff := TRUE;
            MagazinVacuumOn := FALSE;
            CraneTurnCounterclockwise := FALSE;
            CraneTurnClockwise := FALSE;
            StartVar := FALSE;
            StartCommandCrane := FALSE;
            IF (StartButtonMagazin = TRUE) THEN
                interconnectCraneStartCommand := TRUE;
            END_IF;
            IF interconnectCraneStartCommand THEN
                Transit := TRUE;
                State := Crane_states_t#Crane_Init;
            END_IF;

        Crane_states_t#Step0:
            Transit := FALSE;
            IF NOT MagazinCapacitiveSensor THEN
                Transit := TRUE;
                State := Crane_states_t#Crane_Lift_Magazin;
            ELSIF MagazinCapacitiveSensor THEN
                Transit := TRUE;
                State := Crane_states_t#Crane_Lift_Magazin_Metallic;
            END_IF;

        Crane_states_t#Step2:
            Transit := FALSE;
            IF TRUE THEN
                Transit := TRUE;
                State := Crane_states_t#Start_Crane;
            END_IF;

        Crane_states_t#Suck_At_Stamp:
            Transit := FALSE;
            MagazinVacuumOn := TRUE;
            MagazinVacuumOff := FALSE;
            IF CraneSucked THEN
                Transit := TRUE;
                State := Crane_states_t#Crane_Lift_At_Stamp;
            END_IF;

        Crane_states_t#TimeDelay:
            Transit := FALSE;
            TimeDelay_Timer(IN := TRUE, PT := TimeDelay_Timer_Duration);
            TimeDelay_Timer_interconnect := TimeDelay_Timer.Q;
            IF TimeDelay_Timer_interconnect THEN
                Transit := TRUE;
                State := Crane_states_t#Turn_Right;
            END_IF;

        Crane_states_t#Turn_Right:
            Transit := FALSE;
            CraneTurnClockwise := TRUE;
            CraneTurnCounterclockwise := FALSE;
            IF CraneOnMagazin THEN
                Transit := TRUE;
                State := Crane_states_t#Interstep_Check_Workpiece;
            END_IF;

        Crane_states_t#Wait_At_Stamp:
            Transit := FALSE;
            IF TRUE THEN
                Transit := TRUE;
                State := Crane_states_t#pause;
            END_IF;

        Crane_states_t#pause:
            Transit := FALSE;
            Timer1(IN := CraneUp, PT := Duration1);
            interconnect := Timer1.Q;
            IF interconnect THEN
                Transit := TRUE;
                State := Crane_states_t#Reset_interconnect;
            END_IF;

        Crane_states_t#release:
            Transit := FALSE;
            MagazinVacuumOff := TRUE;
            MagazinVacuumOn := FALSE;
            IF TRUE THEN
                Transit := TRUE;
                State := Crane_states_t#Crane_Lift_Conveyor;
            END_IF;

        Crane_states_t#release_Workpiece:
            Transit := FALSE;
            MagazinVacuumOff := TRUE;
            MagazinVacuumOn := FALSE;
            IF TRUE THEN
                Transit := TRUE;
                State := Crane_states_t#Crane_Go_Up;
            END_IF;
    END_CASE;
END_FUNCTION_BLOCK

FUNCTION_BLOCK Magazin
    VAR_INPUT  CraneDown : BOOL; END_VAR
    VAR_OUTPUT  CraneLower : BOOL; END_VAR
    VAR_INPUT  CraneOnConveyor : BOOL; END_VAR
    VAR_INPUT  CraneOnMagazin : BOOL; END_VAR
    VAR_INPUT  CraneSucked : BOOL; END_VAR
    VAR_OUTPUT  CraneTurnClockwise : BOOL; END_VAR
    VAR_OUTPUT  CraneTurnCounterclockwise : BOOL; END_VAR
    VAR_INPUT  CraneUp : BOOL; END_VAR
    VAR_OUTPUT  MagazinGreenLamp : BOOL; END_VAR
    VAR_OUTPUT  MagazinSlider : BOOL; END_VAR
    VAR_OUTPUT  MagazinVacuumOff : BOOL; END_VAR
    VAR_OUTPUT  MagazinVacuumOn : BOOL; END_VAR
    VAR_OUTPUT  MagazinWhiteLamp : BOOL; END_VAR
    VAR  SFCInit : BOOL; END_VAR
    VAR_INPUT  SFCReset : BOOL; END_VAR
    VAR_INPUT  SliderMovedOut : BOOL; END_VAR
    VAR_INPUT  SliderNotMovedOut : BOOL; END_VAR
    VAR_INPUT  StartButtonMagazin : BOOL; END_VAR
    VAR_OUTPUT  StartCommandMagazin : BOOL; END_VAR
    VAR_INPUT  StartVar : BOOL; END_VAR
    VAR_INPUT  WorkpieceReady : BOOL; END_VAR
    VAR  State : Magazin_states_t; END_VAR
    VAR Transit : BOOL; END_VAR
    VAR  interconnectMagazinStartCommand : BOOL; END_VAR

    CASE State OF
        Magazin_states_t#Green_Lamp:

            (* begin(onEntry) *)
           Transit := FALSE;
            (* end(onEntry) *)
            (* begin(onActive) *)
            MagazinGreenLamp := TRUE;
            interconnectMagazinStartCommand := FALSE;
            (* end(onActive) *)
            (* begin(transition) *)
            IF TRUE THEN
               Transit := TRUE;
                State := Magazin_states_t#Magazin_Init;
            END_IF;
            (* end(transition) *)
            (* begin(onExit) *)
            (* end(onExit) *)
            (* end(State) *)

        Magazin_states_t#Init:

            (* begin(onEntry) *)
           Transit := FALSE;
            (* end(onEntry) *)
            (* begin(onActive) *)
            (* end(onActive) *)
            (* begin(transition) *)
            IF TRUE THEN
               Transit := TRUE;
                State := Magazin_states_t#Start_Magazin;
            END_IF;
            (* end(transition) *)
            (* begin(onExit) *)
            (* end(onExit) *)
            (* end(State) *)

        Magazin_states_t#Interstep:

            (* begin(onEntry) *)
           Transit := FALSE;
            (* end(onEntry) *)
            (* begin(onActive) *)
            StartCommandMagazin := TRUE;
            (* end(onActive) *)
            (* begin(transition) *)
            IF StartVar THEN
               Transit := TRUE;
                State := Magazin_states_t#convey;
            END_IF;
            (* end(transition) *)
            (* begin(onExit) *)
            (* end(onExit) *)
            (* end(State) *)

        Magazin_states_t#Magazin_Init:

            (* begin(onEntry) *)
           Transit := FALSE;
            (* end(onEntry) *)
            (* begin(onActive) *)
            MagazinSlider := TRUE;
            (* end(onActive) *)
            (* begin(transition) *)
            IF TRUE THEN
               Transit := TRUE;
                State := Magazin_states_t#Magazin_Init_2;
            END_IF;
            (* end(transition) *)
            (* begin(onExit) *)
            (* end(onExit) *)
            (* end(State) *)

        Magazin_states_t#Magazin_Init_2:

            (* begin(onEntry) *)
           Transit := FALSE;
            (* end(onEntry) *)
            (* begin(onActive) *)
            MagazinSlider := FALSE;
            (* end(onActive) *)
            (* begin(transition) *)
            IF TRUE THEN
               Transit := TRUE;
                State := Magazin_states_t#Interstep;
            END_IF;
            (* end(transition) *)
            (* begin(onExit) *)
            (* end(onExit) *)
            (* end(State) *)

        Magazin_states_t#Slider_Move_Back:

            (* begin(onEntry) *)
           Transit := FALSE;
            (* end(onEntry) *)
            (* begin(onActive) *)
            IF ((SliderMovedOut = TRUE) AND (SliderNotMovedOut = FALSE)) THEN
                MagazinSlider := FALSE;
            END_IF;
            (* end(onActive) *)
            (* begin(transition) *)
            IF CraneUp THEN
               Transit := TRUE;
                State := Magazin_states_t#Step1;
            END_IF;
            (* end(transition) *)
            (* begin(onExit) *)
            (* end(onExit) *)
            (* end(State) *)

        Magazin_states_t#Start_Magazin:

            (* begin(onEntry) *)
           Transit := FALSE;
            (* end(onEntry) *)
            (* begin(onActive) *)
            MagazinSlider := FALSE;
            MagazinGreenLamp := FALSE;
            StartVar := FALSE;
            StartCommandMagazin := FALSE;
            IF (StartButtonMagazin = TRUE) THEN
                interconnectMagazinStartCommand := TRUE;
            END_IF;
            (* end(onActive) *)
            (* begin(transition) *)
            IF interconnectMagazinStartCommand THEN
               Transit := TRUE;
                State := Magazin_states_t#Green_Lamp;
            END_IF;
            (* end(transition) *)
            (* begin(onExit) *)
            (* end(onExit) *)
            (* end(State) *)

        Magazin_states_t#Step0:

            (* begin(onEntry) *)
           Transit := FALSE;
            (* end(onEntry) *)
            (* begin(onActive) *)
            (* end(onActive) *)
            (* begin(transition) *)
            IF CraneDown THEN
               Transit := TRUE;
                State := Magazin_states_t#Slider_Move_Back;
            END_IF;
            (* end(transition) *)
            (* begin(onExit) *)
            (* end(onExit) *)
            (* end(State) *)

        Magazin_states_t#Step1:

            (* begin(onEntry) *)
           Transit := FALSE;
            (* end(onEntry) *)
            (* begin(onActive) *)
            (* end(onActive) *)
            (* begin(transition) *)
            IF CraneOnConveyor THEN
               Transit := TRUE;
                State := Magazin_states_t#Interstep;
            END_IF;
            (* end(transition) *)
            (* begin(onExit) *)
            (* end(onExit) *)
            (* end(State) *)

        Magazin_states_t#convey:

            (* begin(onEntry) *)
           Transit := FALSE;
            (* end(onEntry) *)
            (* begin(onActive) *)
            IF SliderNotMovedOut THEN
                MagazinSlider := TRUE;
            END_IF;
            (* end(onActive) *)
            (* begin(transition) *)
            IF CraneOnMagazin THEN
               Transit := TRUE;
                State := Magazin_states_t#Step0;
            END_IF;
            (* end(transition) *)
            (* begin(onExit) *)
            (* end(onExit) *)
            (* end(State) *)

            END_CASE;
END_FUNCTION_BLOCK

FUNCTION_BLOCK Stamp
    VAR_INPUT  CraneDown : BOOL; END_VAR (*Irwxp*)
    VAR_INPUT  CraneOnConveyor : BOOL; END_VAR (*Irwxp*)
    VAR_INPUT  CranePositionStamp : BOOL; END_VAR (*Irwxp*)
    VAR_INPUT  CraneSucked : BOOL; END_VAR (*Irwxp*)
    VAR_INPUT  CraneUp : BOOL; END_VAR (*Irwxp*)
    VAR  Duration : TIME := TIME#500.0ms; END_VAR (*Lrwxp*)
    VAR  SFCInit : BOOL; END_VAR (*Lrwxp*)
    VAR_INPUT  SFCReset : BOOL; END_VAR (*Irwxp*)
    VAR_OUTPUT  StampGreenLamp : BOOL; END_VAR (*Orwxp*)
    VAR_INPUT  StampLowered : BOOL; END_VAR (*Irwxp*)
    VAR_OUTPUT  StampPressure : BOOL; END_VAR (*Orwxp*)
    VAR_OUTPUT  StampPusher : BOOL; END_VAR (*Orwxp*)
    VAR_INPUT  StampSliderFilled : BOOL; END_VAR (*Irwxp*)
    VAR_OUTPUT  StampSliderMovedIn : BOOL; END_VAR (*Orwxp*)
    VAR_OUTPUT  StampSliderMovedOut : BOOL; END_VAR (*Orwxp*)
    VAR_INPUT  StampSliderSensorMovedIn : BOOL; END_VAR (*Irwxp*)
    VAR_INPUT  StampSliderSensorMovedOut : BOOL; END_VAR (*Irwxp*)
    VAR_INPUT  StampStartButton : BOOL; END_VAR (*Irwxp*)
    VAR_INPUT  StampUp : BOOL; END_VAR (*Irwxp*)
    VAR_OUTPUT  StampWhiteLamp : BOOL; END_VAR (*Orwxp*)
    VAR_OUTPUT  StartCommandStamp : BOOL; END_VAR (*Orwxp*)
    VAR_INPUT  StartVar : BOOL; END_VAR (*Irwxp*)
    VAR  Timer : TON; END_VAR (*Lrwxp*)
    VAR  State : Stamp_states_t; END_VAR (*Lrwxp*)
    VAR  Transit : BOOL; END_VAR (*Lrwxp*)
    VAR  interconnect : BOOL; END_VAR (*Lrwxp*)
    VAR  interconnectStampStartCommand : BOOL; END_VAR (*Lrwxp*)

    CASE State OF
        Stamp_states_t#Green_Lamp:

            (* begin(onEntry) *)
            Transit := FALSE;
            (* end(onEntry) *)
            (* begin(onActive) *)
            StampGreenLamp := TRUE;
            interconnectStampStartCommand := FALSE;
            (* end(onActive) *)
            (* begin(transition) *)
            IF TRUE THEN
                Transit := TRUE;
                State := Stamp_states_t#Stamp_Init_1;
            END_IF;
            (* end(transition) *)
            (* begin(onExit) *)
            (* end(onExit) *)
            (* end(State) *)

        Stamp_states_t#Init:

            (* begin(onEntry) *)
            Transit := FALSE;
            (* end(onEntry) *)
            (* begin(onActive) *)
            (* end(onActive) *)
            (* begin(transition) *)
            IF TRUE THEN
                Transit := TRUE;
                State := Stamp_states_t#Start_Stamp;
            END_IF;
            (* end(transition) *)
            (* begin(onExit) *)
            (* end(onExit) *)
            (* end(State) *)

        Stamp_states_t#Interstep:

            (* begin(onEntry) *)
            Transit := FALSE;
            (* end(onEntry) *)
            (* begin(onActive) *)
            StartCommandStamp := TRUE;
            (* end(onActive) *)
            (* begin(transition) *)
            IF StartVar THEN
                Transit := TRUE;
                State := Stamp_states_t#Interstep_2;
            END_IF;
            (* end(transition) *)
            (* begin(onExit) *)
            (* end(onExit) *)
            (* end(State) *)

        Stamp_states_t#Interstep_2:

            (* begin(onEntry) *)
            Transit := FALSE;
            (* end(onEntry) *)
            (* begin(onActive) *)
            (* end(onActive) *)
            (* begin(transition) *)
            IF StampSliderFilled THEN
                Transit := TRUE;
                State := Stamp_states_t#Step0;
            END_IF;
            (* end(transition) *)
            (* begin(onExit) *)
            (* end(onExit) *)
            (* end(State) *)

        Stamp_states_t#StampProcess:

            (* begin(onEntry) *)
            Transit := FALSE;
            (* end(onEntry) *)
            (* begin(onActive) *)
            StampSliderMovedIn := FALSE;
            StampPusher := TRUE;
            (* end(onActive) *)
            (* begin(transition) *)
            IF StampLowered THEN
                Transit := TRUE;
                State := Stamp_states_t#Step1;
            END_IF;
            (* end(transition) *)
            (* begin(onExit) *)
            (* end(onExit) *)
            (* end(State) *)

        Stamp_states_t#StampSliderBack:

            (* begin(onEntry) *)
            Transit := FALSE;
            (* end(onEntry) *)
            (* begin(onActive) *)
            StampSliderMovedIn := TRUE;
            StampSliderMovedOut := FALSE;
            (* end(onActive) *)
            (* begin(transition) *)
            IF StampSliderSensorMovedIn THEN
                Transit := TRUE;
                State := Stamp_states_t#StampProcess;
            END_IF;
            (* end(transition) *)
            (* begin(onExit) *)
            (* end(onExit) *)
            (* end(State) *)

        Stamp_states_t#StampSliderForward:

            (* begin(onEntry) *)
            Transit := FALSE;
            (* end(onEntry) *)
            (* begin(onActive) *)
            StampPusher := FALSE;
            StampSliderMovedOut := TRUE;
            IF ((StampLowered = FALSE) AND (StampUp = TRUE)) THEN
                interconnect := FALSE;
            END_IF;
            Timer(IN := FALSE, PT := TIME#1.0ms);
            (* end(onActive) *)
            (* begin(transition) *)
            IF StampSliderMovedOut THEN
                Transit := TRUE;
                State := Stamp_states_t#Step2;
            END_IF;
            (* end(transition) *)
            (* begin(onExit) *)
            (* end(onExit) *)
            (* end(State) *)

        Stamp_states_t#Stamp_Init_1:

            (* begin(onEntry) *)
            Transit := FALSE;
            (* end(onEntry) *)
            (* begin(onActive) *)
            StampSliderMovedIn := TRUE;
            StampSliderMovedOut := FALSE;
            (* end(onActive) *)
            (* begin(transition) *)
            IF StampSliderSensorMovedIn THEN
                Transit := TRUE;
                State := Stamp_states_t#Stamp_Init_2;
            END_IF;
            (* end(transition) *)
            (* begin(onExit) *)
            (* end(onExit) *)
            (* end(State) *)

        Stamp_states_t#Stamp_Init_2:

            (* begin(onEntry) *)
            Transit := FALSE;
            (* end(onEntry) *)
            (* begin(onActive) *)
            StampSliderMovedIn := FALSE;
            StampSliderMovedOut := TRUE;
            (* end(onActive) *)
            (* begin(transition) *)
            IF StampSliderSensorMovedOut THEN
                Transit := TRUE;
                State := Stamp_states_t#Stamp_Init_3;
            END_IF;
            (* end(transition) *)
            (* begin(onExit) *)
            (* end(onExit) *)
            (* end(State) *)

        Stamp_states_t#Stamp_Init_3:

            (* begin(onEntry) *)
            Transit := FALSE;
            (* end(onEntry) *)
            (* begin(onActive) *)
            StampPusher := TRUE;
            (* end(onActive) *)
            (* begin(transition) *)
            IF StampLowered THEN
                Transit := TRUE;
                State := Stamp_states_t#Stamp_Init_4;
            END_IF;
            (* end(transition) *)
            (* begin(onExit) *)
            (* end(onExit) *)
            (* end(State) *)

        Stamp_states_t#Stamp_Init_4:

            (* begin(onEntry) *)
            Transit := FALSE;
            (* end(onEntry) *)
            (* begin(onActive) *)
            StampPusher := FALSE;
            (* end(onActive) *)
            (* begin(transition) *)
            IF StampUp THEN
                Transit := TRUE;
                State := Stamp_states_t#Interstep;
            END_IF;
            (* end(transition) *)
            (* begin(onExit) *)
            (* end(onExit) *)
            (* end(State) *)

        Stamp_states_t#Start_Stamp:

            (* begin(onEntry) *)
            Transit := FALSE;
            (* end(onEntry) *)
            (* begin(onActive) *)
            StampSliderMovedOut := FALSE;
            StampSliderMovedIn := FALSE;
            StampPusher := FALSE;
            StampGreenLamp := FALSE;
            StampPressure := FALSE;
            StartCommandStamp := FALSE;
            IF (StampStartButton = TRUE) THEN
                interconnectStampStartCommand := TRUE;
            END_IF;
            (* end(onActive) *)
            (* begin(transition) *)
            IF interconnectStampStartCommand THEN
                Transit := TRUE;
                State := Stamp_states_t#Green_Lamp;
            END_IF;
            (* end(transition) *)
            (* begin(onExit) *)
            (* end(onExit) *)
            (* end(State) *)

        Stamp_states_t#Step0:

            (* begin(onEntry) *)
            Transit := FALSE;
            (* end(onEntry) *)
            (* begin(onActive) *)
            (* end(onActive) *)
            (* begin(transition) *)
            IF CraneUp THEN
                Transit := TRUE;
                State := Stamp_states_t#StampSliderBack;
            END_IF;
            (* end(transition) *)
            (* begin(onExit) *)
            (* end(onExit) *)
            (* end(State) *)

        Stamp_states_t#Step1:

            (* begin(onEntry) *)
            Transit := FALSE;
            (* end(onEntry) *)
            (* begin(onActive) *)
            Timer(IN := StampLowered, PT := T#500ms);
            interconnect := Timer.Q;
            (* end(onActive) *)
            (* begin(transition) *)
            IF interconnect THEN
                Transit := TRUE;
                State := Stamp_states_t#StampSliderForward;
            END_IF;
            (* end(transition) *)
            (* begin(onExit) *)
            (* end(onExit) *)
            (* end(State) *)

        Stamp_states_t#Step2:

            (* begin(onEntry) *)
            Transit := FALSE;
            (* end(onEntry) *)
            (* begin(onActive) *)
            (* end(onActive) *)
            (* begin(transition) *)
            IF CraneOnConveyor THEN
                Transit := TRUE;
                State := Stamp_states_t#Interstep;
            END_IF;
            (* end(transition) *)
            (* begin(onExit) *)
            (* end(onExit) *)
            (* end(State) *)

            END_CASE;
END_FUNCTION_BLOCK

TYPE
    Stamp_states_t : (Green_Lamp , Init , Interstep , Interstep_2 , StampProcess , StampSliderBack , StampSliderForward , Stamp_Init_1 , Stamp_Init_2 , Stamp_Init_3 , Stamp_Init_4 , Start_Stamp , Step0 , Step1 , Step2);
    Magazin_states_t : (Green_Lamp , Init , Interstep , Magazin_Init , Magazin_Init_2 , Slider_Move_Back , Start_Magazin , Step0 , Step1 , convey);
    Crane_states_t : (Crane_Go_Up , Crane_Init , Crane_Init_2 , Crane_Lift_At_Stamp , Crane_Lift_Conveyor , Crane_Lift_Magazin , Crane_Lift_Magazin_Metallic , Crane_Lower , Crane_On_Conveyor , Crane_On_Conveyor_Metallic , Crane_On_Stamp_Metallic , Crane_Turn_Left_From_Stamp , Crane_Turn_Left_Metallic , Crane_Turn_Left_NOT_Metallic , Init , Interstep , Interstep_2 , Interstep_Check_Workpiece , Lower_Crane , Reset_interconnect , Start_Crane , Step0 , Step2 , Suck_At_Stamp , TimeDelay , Turn_Right , Wait_At_Stamp , pause , release , release_Workpiece);
END_TYPE

FUNCTION_BLOCK TON
VAR_INPUT
  IN : BOOL;
  PT : TIME;
END_VAR
VAR
  running : BOOL;
END_VAR
VAR_TEMP
    timeout : BOOL;
END_VAR
VAR_OUTPUT
  Q : BOOL;
  ET : TIME;
END_VAR
  timeout := NONDETERMINISTIC_BOOL();
  IF NOT IN THEN
    Q := FALSE;
    running := FALSE;
  ELSIF NOT running AND NOT Q THEN
    running := TRUE;
  ELSIF running AND NOT Q THEN
    Q := timeout;
    running := NOT Q;
  END_IF;

  ET := NONDETERMINISTIC_TIME();
END_FUNCTION_BLOCK

(* ---- Scenario3v1_Final_Main.st ---- *)
PROGRAM Main

VAR  Actuator_AnalogCranePressure : INT; END_VAR (*Lrwxp*)
VAR  Actuator_CraneLower : BOOL; END_VAR (*Lrwxp*)
VAR  Actuator_CraneTurnClockwise : BOOL; END_VAR (*Lrwxp*)
VAR  Actuator_CraneTurnCounterclockwise : BOOL; END_VAR (*Lrwxp*)
VAR  Actuator_MagazinGreenLamp : BOOL; END_VAR (*Lrwxp*)
VAR  Actuator_MagazinSlider : BOOL; END_VAR (*Lrwxp*)
VAR  Actuator_MagazinVacuumOff : BOOL; END_VAR (*Lrwxp*)
VAR  Actuator_MagazinVacuumOn : BOOL; END_VAR (*Lrwxp*)
VAR  Actuator_MagazinWhiteLamp : BOOL; END_VAR (*Lrwxp*)
VAR  Actuator_SomeActuator : BOOL; END_VAR (*Lrwxp*)
VAR  Actuator_StampGreenLamp : BOOL; END_VAR (*Lrwxp*)
VAR  Actuator_StampPusher : BOOL; END_VAR (*Lrwxp*)
VAR  Actuator_StampSliderMovedIn : BOOL; END_VAR (*Lrwxp*)
VAR  Actuator_StampSliderMovedOut : BOOL; END_VAR (*Lrwxp*)
VAR  Actuator_StampWhiteLamp : BOOL; END_VAR (*Lrwxp*)
VAR  Crane : Crane; END_VAR (*Lrwxp*)
VAR  Mag : Magazin; END_VAR (*Lrwxp*)
VAR  Sensor_CraneDown : BOOL; END_VAR (*Lrwxp*)
VAR  Sensor_CraneOnConveyor : BOOL; END_VAR (*Lrwxp*)
VAR  Sensor_CraneOnMagazin : BOOL; END_VAR (*Lrwxp*)
VAR  Sensor_CranePosition : BOOL; END_VAR (*Lrwxp*)
VAR  Sensor_CranePositionStamp : BOOL; END_VAR (*Lrwxp*)
VAR  Sensor_CraneSucked : BOOL; END_VAR (*Lrwxp*)
VAR  Sensor_CraneUp : BOOL; END_VAR (*Lrwxp*)
VAR  Sensor_MagazinCapacitiveSensor : BOOL; END_VAR (*Lrwxp*)
VAR  Sensor_MagazinEmergencyStop : BOOL; END_VAR (*Lrwxp*)
VAR  Sensor_MagazinOpticalSensor : BOOL; END_VAR (*Lrwxp*)
VAR  Sensor_MagazinSwitchManuellAutomatic : BOOL; END_VAR (*Lrwxp*)
VAR  Sensor_SliderMovedOut : BOOL; END_VAR (*Lrwxp*)
VAR  Sensor_SliderNotMovedOut : BOOL; END_VAR (*Lrwxp*)
VAR  Sensor_StampEmergencyStop : BOOL; END_VAR (*Lrwxp*)
VAR  Sensor_StampLowered : BOOL; END_VAR (*Lrwxp*)
VAR  Sensor_StampSliderFilled : BOOL; END_VAR (*Lrwxp*)
VAR  Sensor_StampSliderSensorMovedIn : BOOL; END_VAR (*Lrwxp*)
VAR  Sensor_StampSliderSensorMovedOut : BOOL; END_VAR (*Lrwxp*)
VAR  Sensor_StampStartButton : BOOL; END_VAR (*Lrwxp*)
VAR  Sensor_StampSwitchManuellAutomatic : BOOL; END_VAR (*Lrwxp*)
VAR  Sensor_StampUp : BOOL; END_VAR (*Lrwxp*)
VAR  Sensor_StartButtonMagazin : BOOL; END_VAR (*Lrwxp*)
VAR  Sensor_WorkpieceReady : BOOL; END_VAR (*Lrwxp*)
VAR  Stamp : Stamp; END_VAR (*Lrwxp*)
Mag.SliderNotMovedOut := Sensor_SliderNotMovedOut;
Mag.SliderMovedOut := Sensor_SliderMovedOut;
Mag.CraneOnMagazin := Sensor_CraneOnMagazin;
Mag.CraneDown := Sensor_CraneDown;
Mag.CraneUp := Sensor_CraneUp;
Mag.CraneOnConveyor := Sensor_CraneOnConveyor;
Mag.WorkpieceReady := Sensor_WorkpieceReady;
Mag.StartButtonMagazin := Sensor_StartButtonMagazin;
Actuator_MagazinSlider := Mag.MagazinSlider;
Actuator_MagazinGreenLamp := Mag.MagazinGreenLamp;
Crane.CraneUp := Sensor_CraneUp;
Crane.CraneOnConveyor := Sensor_CraneOnConveyor;
Crane.CraneDown := Sensor_CraneDown;
Crane.CraneSucked := Sensor_CraneSucked;
Crane.CraneOnMagazin := Sensor_CraneOnMagazin;
Crane.MagazinCapacitiveSensor := Sensor_MagazinCapacitiveSensor;
Crane.CranePositionStamp := Sensor_CranePositionStamp;
Crane.SliderMovedOut := Sensor_SliderMovedOut;
Crane.WorkpieceReady := Sensor_WorkpieceReady;
Crane.StampSliderFilled := Sensor_StampSliderFilled;
Crane.SliderMovedOut := Sensor_SliderMovedOut;
Crane.StartButtonMagazin := Sensor_StartButtonMagazin;
Actuator_CraneTurnCounterclockwise := Crane.CraneTurnCounterclockwise;
Actuator_CraneTurnClockwise := Crane.CraneTurnClockwise;
Actuator_CraneLower := Crane.CraneLower;
Actuator_MagazinVacuumOff := Crane.MagazinVacuumOff;
Actuator_MagazinVacuumOn := Crane.MagazinVacuumOn;
Stamp.StampSliderSensorMovedOut := Sensor_StampSliderSensorMovedOut;
Stamp.StampSliderSensorMovedIn := Sensor_StampSliderSensorMovedIn;
Stamp.StampSliderFilled := Sensor_StampSliderFilled;
Stamp.StampUp := Sensor_StampUp;
Stamp.StampLowered := Sensor_StampLowered;
Stamp.CraneDown := Sensor_CraneDown;
Stamp.CraneUp := Sensor_CraneUp;
Stamp.CraneSucked := Sensor_CraneSucked;
Stamp.CranePositionStamp := Sensor_CranePositionStamp;
Stamp.CraneOnConveyor := Sensor_CraneOnConveyor;
Stamp.StampStartButton := Sensor_StampStartButton;
Actuator_StampSliderMovedOut := Stamp.StampSliderMovedOut;
Actuator_StampSliderMovedIn := Stamp.StampSliderMovedIn;
Actuator_StampWhiteLamp := Stamp.StampWhiteLamp;
Actuator_StampPusher := Stamp.StampPusher;
Actuator_StampGreenLamp := Stamp.StampGreenLamp;
Actuator_AnalogCranePressure := INT#6000;
IF (Sensor_StampEmergencyStop AND Sensor_MagazinEmergencyStop) THEN
    Mag();
    Crane();
    Stamp();
    IF (Actuator_MagazinGreenLamp AND Actuator_StampGreenLamp) THEN
        IF ((Stamp.StartCommandStamp AND Crane.StartCommandCrane) AND Mag.StartCommandMagazin) THEN
            Crane.StartVar := TRUE;
            Mag.StartVar := TRUE;
            Stamp.StartVar := TRUE;
        END_IF;
    END_IF;
    Crane.SFCReset := FALSE;
    Mag.SFCReset := FALSE;
    Stamp.SFCReset := FALSE;
ELSIF (NOT Sensor_StampEmergencyStop OR NOT Sensor_MagazinEmergencyStop) THEN
    Actuator_MagazinSlider := FALSE;
    Actuator_CraneLower := FALSE;
    Actuator_MagazinVacuumOn := FALSE;
    Actuator_MagazinVacuumOff := TRUE;
    Actuator_MagazinGreenLamp := FALSE;
    Actuator_CraneTurnCounterclockwise := FALSE;
    Actuator_CraneTurnClockwise := FALSE;
    Actuator_StampSliderMovedOut := TRUE;
    Actuator_StampSliderMovedIn := FALSE;
    Actuator_StampGreenLamp := FALSE;
    Actuator_StampPusher := FALSE;
    Actuator_AnalogCranePressure := INT#0;
    Crane.SFCReset := TRUE;
    Mag.SFCReset := TRUE;
    Stamp.SFCReset := TRUE;
    Crane.StartVar := FALSE;
    Mag.StartVar := FALSE;
    Stamp.StartVar := FALSE;
END_IF;
END_PROGRAM
